(* IEC 61131-3 sources: iFA_git_test/GIT test/PLC_1/Programs, 4 files *)

(* ---- DefaultVariableTable.st ---- *)
(*NodeCRC64:15794442468608431415, FileCRC64:15258916066108261974*)
VAR_GLOBAL
END_VAR

(*{"Version":"1.0.0.0","Path":"Default_variable_table","ObjectType":"Global"}*)

END_VAR_GLOBAL

(* ---- FB_Example.st ---- *)
(*NodeCRC64:9907401017642776752, FileCRC64:7915297945421370368*)
FUNCTION_BLOCK FB_Example
VAR_INPUT
END_VAR
VAR_OUTPUT
END_VAR
VAR
END_VAR

Body

EndBody

(*{"Version":"1.0.0.0","Path":"FB_Example","ObjectType":"FunctionBlock"}*)

END_FUNCTION_BLOCK

(* ---- FB_LowPass.st ---- *)
(*NodeCRC64:0, FileCRC64:0*)
FUNCTION_BLOCK FB_LowPass
VAR_INPUT
    lrInput : LREAL;
    lrCutoffFreq : LREAL;
    lrSampleTime : LREAL;
END_VAR
VAR_OUTPUT
    lrOutput : LREAL;
END_VAR
VAR
    lrAlpha : LREAL;
END_VAR

Body
    IF lrCutoffFreq > 0.0 AND lrSampleTime > 0.0 THEN
        lrAlpha := lrSampleTime /
                   (lrSampleTime + (1.0 / (2.0 * 3.14159265359 * lrCutoffFreq)));

        lrOutput := lrOutput + lrAlpha * (lrInput - lrOutput);
    ELSE
        lrOutput := lrInput;
    END_IF;
EndBody

(*{"Version":"1.0.0.0","Path":"FB_LowPass","ObjectType":"FunctionBlock"}*)

END_FUNCTION_BLOCK

(* ---- Main.st ---- *)
(*NodeCRC64:12862529608055231842, FileCRC64:3733895348766379544*)
PROGRAM Main
VAR
    liCounter : LINT;
END_VAR

Body
liCounter := liCounter + 1;
EndBody

(*{"Version":"1.0.0.0","Path":"Main","ObjectType":"Program"}*)

END_PROGRAM
